(********************* G.D S.p.A. - Technical Department ***********************************
This program has been generated automatically from Application Designer DE&F
********************************************************************************************)
PROGRAM dbg_csp_transfer_upstacker_sensors
VAR
  carton_backstop_di_shd : digital_input_shadow;
  prime_di_shd : digital_input_shadow;
END_VAR

_objects_manager();

IF	g_application_status <> APPLICATION_STATUS_RUNNING
THEN
	RETURN;
END_IF

CASE process_get_mode(CONVERSION_this := dbg_root.prc) OF
	MODE_ABSENT,
	MODE_INACTIVE:
		RETURN;
	MODE_TEST:
		RETURN;
END_CASE

ACTION _objects_manager:
IF	objects_initialization()
THEN
	digital_input_shadow_init(
		sim_mode:= SHADOW_SIMULATION_MODE_AUTOMATIC, 
		father:= csp_transfer_upstacker_sensors.carton_backstop_di, 
		process:= dbg_root.prc, 
		CONVERSION_this:= carton_backstop_di_shd);

	digital_input_shadow_init(
		sim_mode:= SHADOW_SIMULATION_MODE_AUTOMATIC, 
		father:= csp_transfer_upstacker_sensors.prime_di, 
		process:= dbg_root.prc, 
		CONVERSION_this:= prime_di_shd);

	RETURN;
END_IF

IF	objects_running()
THEN
	digital_input_shadow_cycle(carton_backstop_di_shd);
	digital_input_shadow_cycle(prime_di_shd);
END_IF
END_ACTION

END_PROGRAM

(* stored: Version 1.1.0.1, ProductVersion 3.1.4022.12
   POU dbg_csp_transfer_upstacker_sensors: Id {d06a7ed9-6f28-4ccb-b89c-6d32260f6359}, SpecialFunc None
   Action _objects_manager: Id {344f9869-65aa-4b61-8db0-a24787e8525c} *)
